{attribute 'call_after_init'}
FUNCTION_BLOCK FB_Arbiter_Test EXTENDS TcUnit.FB_TestSuite
VAR_INPUT
END_VAR
VAR_OUTPUT
END_VAR
VAR
END_VAR

Arbitration();
RequestCheckRemoveBP();
FullArbitrationStack();

METHOD Arbitration
VAR_INPUT
END_VAR
VAR
    
     nAttReqID    :    UDINT    := 1;
    stAttReqBP    :    ST_BeamParams := PMPS_GVL.cstFullBeam;
    
    nPPEReqID    :    UDINT    := 2;
    stPPEReqBP    :    ST_BeamParams := PMPS_GVL.cstFullBeam;
    
    nEVReqID    :    UDINT    := 3;
    stEVReqBP    :    ST_BeamParams := PMPS_GVL.cstFullBeam;
    
    nRateReqID    :    UDINT    := 4;
    stRateReqBP    :    ST_BeamParams := PMPS_GVL.cstFullBeam;
    
    stArbitratedBP    :    ST_BeamParams;
    stExpectedBP    :    ST_BeamParams;
END_VAR
VAR_INST
    fbArbiter    :    FB_Arbiter(1);
END_VAR
TEST('Arbitration');

stAttReqBP.fAtt := 50;
stPPEReqBP.fPP_mJ := 1;
stEVReqBP.neVRange := 2#1111_1100_1111_1111;
stRateReqBP.nRate := 120;

//Load arbiter with beam parameter sets
AssertTrue(fbArbiter.AddRequest(nAttReqID, stAttReqBP),
                    'Safest attenuation request failed to load');
                    
//Load arbiter with beam parameter sets
AssertTrue(fbArbiter.AddRequest(nPPEReqID, stPPEReqBP),
                    'Safest PPE request failed to load');
                    
//Load arbiter with beam parameter sets
AssertTrue(fbArbiter.AddRequest(nEVReqID, stEVReqBP),
                    'Safest stEVReqBP request failed to load');
                    
//Load arbiter with beam parameter sets
AssertTrue(fbArbiter.AddRequest(nRateReqID, stRateReqBP),
                    'Safest stEVReqBP request failed to load');

stExpectedBP.fAtt     :=     stAttReqBP.fAtt;
stExpectedBP.fPP_mJ    :=  stPPEReqBP.fPP_mJ;
stExpectedBP.neVRange := stEVReqBP.neVRange;
stExpectedBP.nRate := stRateReqBP.nRate;

stArbitratedBP := fbArbiter.GetArbitratedBP();

AssertFalse(F_DiffReqBeamParams(stExpectedBP, stArbitratedBP),
                'Arbitrated BP does not match expected.');

TEST_FINISHED();
END_METHOD

METHOD FullArbitrationStack
VAR_INPUT
END_VAR
VAR   
    nId    :    DWORD := 1;
    stReq    :    ST_BeamParams := (fAtt:=12);
END_VAR
VAR_INST
    fbArbiter    :    FB_Arbiter(1);
    
    fbHigherArb : FB_Arbiter(2);
    
    fbSubSysToArb : FB_SubSysToArbiter_IO;
    pBPR : POINTER TO ST_BeamParams;
    fbArbToSubSys : FB_ArbiterToSubSys_IO := (RequestingSystemID:=34);
    pBPC : POINTER TO ST_BeamParams;
    
    fbBPR : FB_BPRequestor;
    
    FFO : FB_HardwareFFOutput;
    
    State : INT := 10;
    testidx : INT := 10;
    Cycle : INT := 0;
    
END_VAR
TEST('FullStack');

fbArbiter.AddRequest(nId, stReq); // some device asking it's arbiter for some beam parameters

TEST('CheckBPNotValidYet');
AssertFalse(fbArbiter.CheckRequest(nId),
    'Check should fail. Request not arbitrated yet.');
TEST_FINISHED();

CASE state OF

10:
    
    
    ///////////////////////////////////////
    //Sub system cycle
    fbSubSysToArb(Arbiter := fbArbiter, fbFFHWO := FFO);
    //END of sub system cycle
    ///////////////////////////////////////
    
    //Ethercat transfer simulation
    pBPR := ADR(fbArbToSubSys.i_RequestedBP);
    pBPR^ := fbSubSysToArb.q_stRequestedBP;
    WRITE_PROTECTED_BOOL(ADR(fbArbToSubSys.i_TxPDOToggle), TRUE);
    
    pBPC := ADR(fbSubSysToArb.i_stCurrentBP);
    pBPC^ := fbArbToSubSys.o_CurrentBP;
    
    //////////////////////////////////////
    //Start of arbiter plc cycle
    //Arb io collects sub system status
    fbArbToSubSys(Arbiter := fbHigherArb, fbFFHWO := FFO);
    //BPR collects arbiter summation
    fbBPR(Arbiter := fbHigherArb);
    
    Cycle := Cycle + 1;
    
    CASE Cycle OF
        2:
            state := 11;
        3:
            state := 12;
        10:
            state := 8000;
    ELSE
        ;
	END_CASE
    
11:
    TEST('CheckBPValidNow');
    AssertTrue(fbArbiter.CheckRequest(nId),
    'Check should pass.');
    TEST_FINISHED_NAMED('CheckBPValidNow');
    
    state := 10;
    
12:
    state := 8000;
    
8000:
    TEST_FINISHED_NAMED('FullStack');
    

END_CASE
END_METHOD

METHOD RequestCheckRemoveBP
VAR_INPUT
END_VAR
VAR
    
    nId    :    DWORD := 1;
    stReq    :    ST_BeamParams;
END_VAR
VAR_INST
    fbArbiter    :    FB_Arbiter(1);
END_VAR
TEST('RequestBP');
AssertTrue(fbArbiter.AddRequest(nId, stReq),
    'Request failed');

TEST_FINISHED();
    
TEST('DuplicateID');
AssertFalse(fbArbiter.AddRequest(nId, stReq),
    'Duplicate request accepted, not good.');

TEST_FINISHED();
    
TEST('CheckBP');
AssertFalse(fbArbiter.CheckRequest(nId),
    'Check should fail. Request not arbitrated yet.');
TEST_FINISHED();

TEST('CheckBPArbitrated');
WRITE_PROTECTED_ULINT(ADR(fbArbiter.nArbiterCohort), fbArbiter.nArbiterCohort + 1);
AssertTrue(fbArbiter.CheckRequest(nId),
    'Check should pass.');

TEST_FINISHED();      
    
TEST('IDDoesNotExist');
WRITE_PROTECTED_ULINT(ADR(fbArbiter.nArbiterCohort), fbArbiter.nArbiterCohort + 1); 
AssertFalse(fbArbiter.CheckRequest(nId+1),
    'Check returned true when ID does not exist');

TEST_FINISHED();
    
TEST('RemoveBP');
AssertTrue(fbArbiter.RemoveRequest(nId),
    'Remove failed');
AssertFalse(fbArbiter.CheckRequest(nId),
    'Remove did not remove request');
    
TEST_FINISHED();
END_METHOD

END_FUNCTION_BLOCK

(* stored: Version 1.1.0.1, ProductVersion 3.1.4022.18
   POU FB_Arbiter_Test: Id {33ac0bc1-5ef2-4a28-bd81-83e3f5956062}, SpecialFunc None
   Method Arbitration: Id {c3caf704-ac1c-41da-98d7-fd2af820601b}
   Method FullArbitrationStack: Id {17fe9309-58be-432c-a642-5a1fae576773}
   Method RequestCheckRemoveBP: Id {62a4c245-663e-41d8-901a-0a0faba360f7} *)
